FUNCTION_BLOCK B_ALGDNC (* Basic Function Block Type *)
  (* Standard: 61499-2 *)
  (* Version 0.0, 2015-11-24, 4DIAC-IDE, 4DIAC-Consortium *)
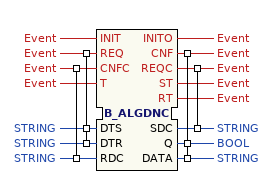
  EVENT_INPUT
    INIT; (* Initialization Request *)
    REQ WITH DTR, DTS; (* Normal Execution Request *)
    CNFC WITH RDC; (* CNF CLIENT *)
    T; (* EO DELAY *)
  END_EVENT
  EVENT_OUTPUT
    INITO; (* Initialization Confirm *)
    CNF WITH Q, DATA; (* Execution Confirmation *)
    REQC WITH SDC; (* REQ CLIENT *)
    ST; (* START DELAY *)
    RT; (* STOP DELAY *)
  END_EVENT
  VAR_INPUT
    DTS : STRING; (* DATA TO SEND *)
    DTR : STRING; (* DATA TO RECIVE *)
    RDC : STRING; (* RD CLIENT *)
  END_VAR
  VAR_OUTPUT
    SDC : STRING; (* SD CLIENT *)
    Q : BOOL; (* RESULT *)
    DATA : STRING;
  END_VAR
  VAR
    OK : BOOL := FALSE; (* Internal Variable *)
    NAK : BOOL := FALSE; (* Internal Variable *)
    NT : UINT := 0; (* Numero Repeticiones DELAY *)
    NE : UINT := 0; (* Numero Repeticones NAKDEL *)
    STRINGNAK : STRING; (* Internal Variable *)
    STX : BOOL := FALSE; (* Internal Variable *)
    STRINGSTX : STRING; (* Internal Variable *)
    STRINGCMP : STRING; (* Internal Variable *)
    EOTDEL : BOOL := FALSE; (* Internal Variable *)
    COMPOSITESTRING : STRING; (* Internal Variable *)
    CMPSTRINGLENGHT : UINT; (* Internal Variable *)
    STRINGETB : STRING; (* Internal Variable *)
    STRINGETX : STRING; (* Internal Variable *)
    TRUNCADA : BOOL := FALSE; (* Internal Variable *)
  END_VAR
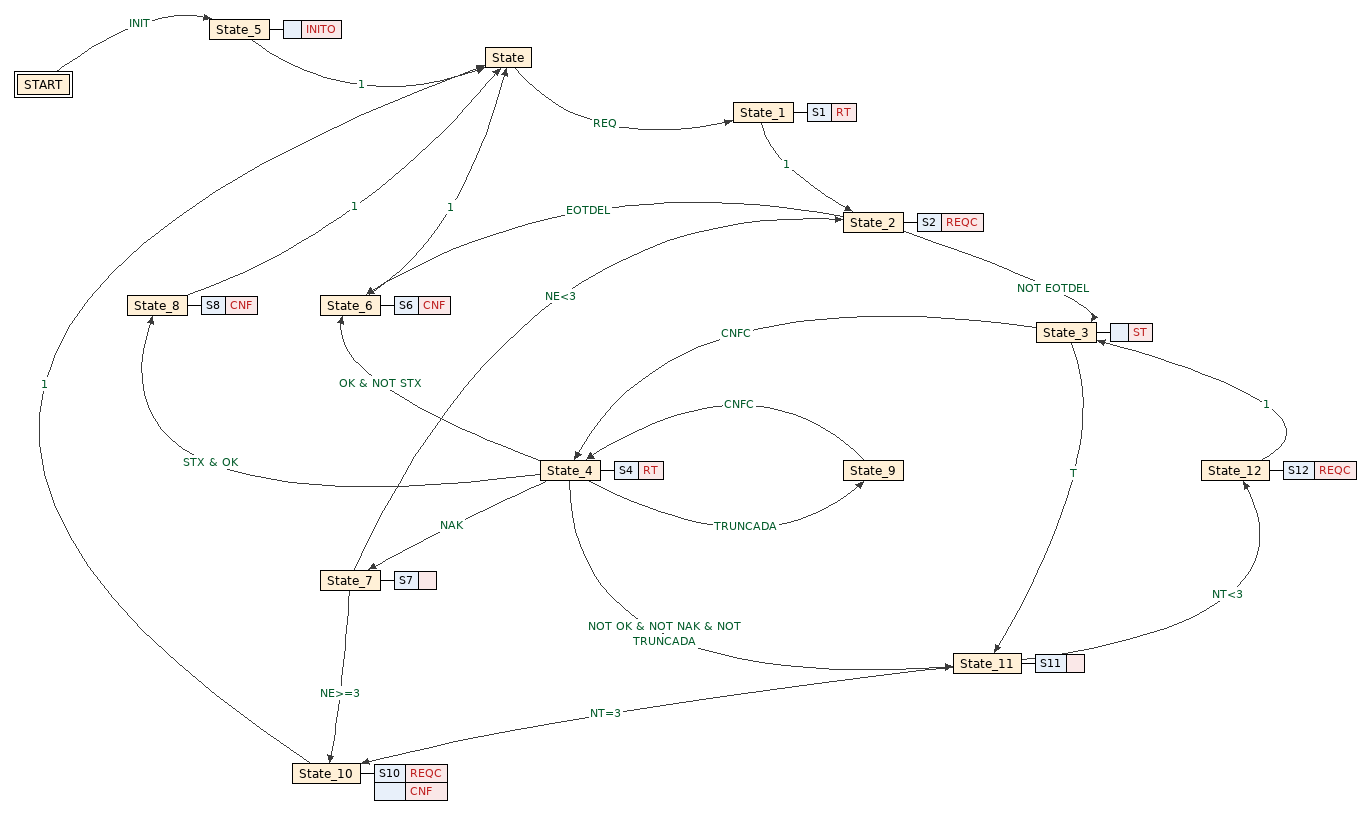
  EC_STATES
    START; (* Initial State *)
    State;
    State_1 : S1 -> RT;
    State_2 : S2 -> REQC;
    State_3 : -> ST;
    State_4 : S4 -> RT;
    State_6 : S6 -> CNF;
    State_7 : S7;
    State_10 : S10 -> REQC, -> CNF;
    State_11 : S11;
    State_12 : S12 -> REQC;
    State_5 : -> INITO;
    State_8 : S8 -> CNF;
    State_9;
  END_STATES
  EC_TRANSITIONS
    State TO State_1 := REQ;
    State_1 TO State_2 := 1;
    State_2 TO State_3 := NOT EOTDEL;
    State_3 TO State_4 := CNFC;
    State_4 TO State_6 := OK & NOT STX;
    State_4 TO State_7 := NAK;
    State_7 TO State_10 := NE>=3;
    State_10 TO State := 1;
    State_11 TO State_10 := NT=3;
    State_11 TO State_12 := NT<3;
    State_6 TO State := 1;
    State_12 TO State_3 := 1;
    State_7 TO State_2 := NE<3;
    State_4 TO State_11 := NOT OK & NOT NAK & NOT TRUNCADA;
    State_3 TO State_11 := T;
    State_2 TO State_6 := EOTDEL;
    START TO State_5 := INIT;
    State_5 TO State := 1;
    State_4 TO State_8 := STX & OK;
    State_8 TO State := 1;
    State_4 TO State_9 := TRUNCADA;
    State_9 TO State_4 := CNFC;
  END_TRANSITIONS
  ALGORITHM INIT IN ST: (* Initialization algorithm *)

  END_ALGORITHM
  ALGORITHM REQ IN ST: (* Normally executed algorithm *)

  END_ALGORITHM
  ALGORITHM S2 IN ST: (* new algorithm *)
SDC:=DTS;
STRINGCMP:='\x01\x02\x03\x04';

IF STRINGCMP=DTR THEN
EOTDEL:=TRUE;
ELSE
EOTDEL:=FALSE;
END_IF;
  END_ALGORITHM
  ALGORITHM S4 IN ST: (* new algorithm *)
STRINGNAK:='\x15\x7f';
STRINGSTX:='\x02';
STRINGETB:='\x17';
STRINGETX:='\x03';
STRINGCMP:= MID(RDC,1,1);




IF RDC=DTR THEN
	OK:=TRUE;
ELSIF RDC=STRINGNAK THEN
	NAK:=TRUE;
ELSE
	NAK:=FALSE;
	OK:=FALSE;
	STX:=FALSE;
END_IF;

IF NOT TRUNCADA THEN
	COMPOSITESTRING:='\x00';
	STRINGCMP:= '\x02\x03';
	IF STRINGCMP=DTR THEN
		STRINGCMP:= MID(RDC,1,1);
		IF STRINGCMP=STRINGSTX THEN
			CMPSTRINGLENGHT:=LEN(RDC)-2;
			STRINGCMP:=MID(RDC,1,CMPSTRINGLENGHT);
			IF STRINGCMP=STRINGETX OR STRINGCMP=STRINGETB THEN
				COMPOSITESTRING:=RDC;
				STX:=TRUE;
				OK:=TRUE;
				TRUNCADA:=FALSE;
			ELSE
				COMPOSITESTRING:=RDC;
				TRUNCADA:=TRUE;
				STX:=FALSE;
				OK:=FALSE;
			END_IF;
		ELSE
			STX:=FALSE;
			OK:=FALSE;
			TRUNCADA:=FALSE;
		END_IF;
	END_IF;
ELSE
	COMPOSITESTRING:=CONCAT(COMPOSITESTRING,RDC);
	CMPSTRINGLENGHT:=LEN(COMPOSITESTRING)-2;
	STRINGCMP:=MID(COMPOSITESTRING,1,CMPSTRINGLENGHT);
	IF STRINGCMP=STRINGETX OR STRINGCMP=STRINGETB THEN
		STX:=TRUE;
		OK:=TRUE;
		TRUNCADA:=FALSE;
	ELSE
		TRUNCADA:=TRUE;
		STX:=FALSE;
		OK:=FALSE;
	END_IF;
END_IF;
  END_ALGORITHM
  ALGORITHM S6 IN ST: (* new algorithm *)
Q:=TRUE;
  END_ALGORITHM
  ALGORITHM S1 IN ST: (* new algorithm *)
NT:=0;
NE:=0;
OK:=FALSE;
NAK:=FALSE;
STX:=FALSE;
EOTDEL:=FALSE;
  END_ALGORITHM
  ALGORITHM S10 IN ST: (* new algorithm *)
SDC:='\x04';
Q:=FALSE;
  END_ALGORITHM
  ALGORITHM S7 IN ST: (* new algorithm *)
NE:=NE+1;
  END_ALGORITHM
  ALGORITHM S11 IN ST: (* new algorithm *)
NT:=NT+1;
  END_ALGORITHM
  ALGORITHM S12 IN ST: (* new algorithm *)
SDC:='\x05';
  END_ALGORITHM
  ALGORITHM S3 IN ST: (* new algorithm *)

  END_ALGORITHM
  ALGORITHM S8 IN ST: (* new algorithm *)
DATA:=COMPOSITESTRING;
Q:=TRUE;
  END_ALGORITHM
END_FUNCTION_BLOCK
